PROGRAM P_Demo_LrealIsFinite
VAR
    lrPidOut : LREAL;; // PID 输出
    bFinite  : BOOL;; // 是否安全使用
    bCheck   : BOOL;
END_VAR

// ============================================================
// Tc2_Utilities.LrealIsFinite 演示程序（FUNCTION，单周期触发）
// ============================================================
// 场景：PID 输出做电机命令前必须先 finite 校验，否则下游 LREAL_TO_INT64 命中 PDF 未定义。
// 价值：替代手写 IEEE 754 位检测；一次调用语义清晰。
// 验证步骤：
//   1. 把本 PROGRAM 加到 PlcTask 调用列表
//   2. 编译 + 登录
//   3. 在线把 b... 触发位置 TRUE 一个周期
//   4. 观察输出变量是否符合期望
// ============================================================

IF bCheck THEN
    // 必须用变量传址 —— REFERENCE TO 不接表达式
    bFinite := LrealIsFinite(lrPidOut);
    bCheck := FALSE;
END_IF;

END_PROGRAM

(* stored: Version 1.1.0.1, ProductVersion 3.1.4024.5
   POU P_Demo_LrealIsFinite: Id {4028b058-3abd-56c1-86d8-70f5a7bb5a3d}, SpecialFunc None *)
